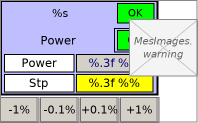
VISUALIZATION VISU_CANON  // 198x123
VAR_IN_OUT
	m_Input_SOURCE : BLOCK_SOURCE_JOULE;
END_VAR
    Rectangle (0,0 158x95)
    Rectangle (3,30 110x21), "Power"
    Rectangle (117,3 37x20), "NOK", invisible if: NOT m_Input_SOURCE.STATE_NOK
    Rectangle (117,30 37x20), "OFF", invisible if: m_Input_SOURCE.STATE_EJ_ON
    Rectangle (117,3 37x20), "OK", invisible if: m_Input_SOURCE.STATE_NOK
    Rectangle (117,30 37x20), "ON", invisible if: NOT m_Input_SOURCE.STATE_EJ_ON
    RoundedRectangle (4,54 70x18), "Power", invisible if: Global_Variables.MACHINE.State_manu
    RoundedRectangle (76,54 77x18), "%.3f %%", text variable: m_Input_SOURCE.STATE_POWER, invisible if: Global_Variables.MACHINE.State_manu
    Rectangle (0,3 120x21), "%s", text variable: m_Input_SOURCE.MNEMO
    Polyline (7,35)
    RoundedRectangle (4,74 70x18), "Stp", invisible if: NOT Global_Variables.PRG_USER.ACTU_USER.MAINTENANCE OR NOT MACHINE.State_manu
    RoundedRectangle (76,74 77x18), "%.3f %%", text variable: m_Input_SOURCE.PRM_POWER, invisible if: NOT Global_Variables.PRG_USER.ACTU_USER.MAINTENANCE OR NOT MACHINE.STATE_Manu
        OnMouseDown: write the text variable via InputWithLimits, min 0, max 100
    Rectangle (114,28 41x24), invisible if: NOT m_Input_SOURCE.EJ.AUTOR_ON_IHM AND NOT m_Input_SOURCE.EJ.AUTOR_Off_IHM, input disabled if: (NOT m_Input_SOURCE.EJ.AUTOR_ON_IHM AND NOT m_Input_SOURCE.EJ.AUTOR_OFF_IHM) OR NOT PRG_User.ACTU_USER.MAINTENANCE
        tap m_Input_SOURCE.EJ.M_On
    Image (129,19 69x57), invisible if: NOT m_Input_SOURCE.STATE_NOK, image: MesImages.warning
    Button (0,97 39x26), "-1%", invisible if: NOT Global_Variables.PRG_USER.ACTU_USER.MAINTENANCE OR NOT MACHINE.STATE_Manu OR (m_Input_SOURCE.PRM_POWER<1.0)
        OnMouseClick: execute { m_Input_SOURCE.PRM_POWER := m_Input_SOURCE.PRM_POWER - 1.0; }
    Button (40,97 39x26), "-0.1%", invisible if: NOT Global_Variables.PRG_USER.ACTU_USER.MAINTENANCE OR NOT MACHINE.STATE_Manu OR (m_Input_SOURCE.PRM_POWER<0.1)
        OnMouseClick: execute { m_Input_SOURCE.PRM_POWER := m_Input_SOURCE.PRM_POWER - 0.1; }
    Button (80,97 39x26), "+0.1%", invisible if: NOT Global_Variables.PRG_USER.ACTU_USER.MAINTENANCE OR NOT MACHINE.STATE_Manu OR (m_Input_SOURCE.PRM_POWER>99.9)
        OnMouseClick: execute { m_Input_SOURCE.PRM_POWER := m_Input_SOURCE.PRM_POWER + 0.1; }
    Button (120,97 39x26), "+1%", invisible if: NOT Global_Variables.PRG_USER.ACTU_USER.MAINTENANCE OR NOT MACHINE.STATE_Manu OR (m_Input_SOURCE.PRM_POWER>99.0)
        OnMouseClick: execute { m_Input_SOURCE.PRM_POWER := m_Input_SOURCE.PRM_POWER + 1.0; }
END_VISUALIZATION

(* stored: Version 1.1.0.1, ProductVersion 3.1.4024.10
   Visu VISU_CANON: Id {78853d43-670a-4e00-8358-f17db1d0e80b} *)
